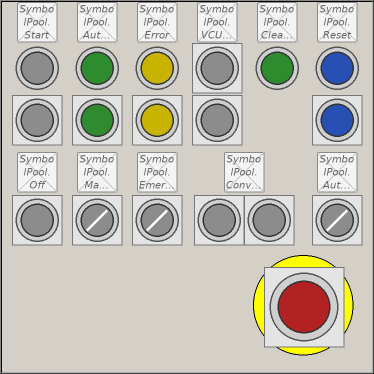
VISUALIZATION V_VC_AccessPanel  // 374x374
VAR_IN_OUT
	Signals : ST_VC_AccessPanel;
END_VAR
    Rectangle (0,0 374x374)
    Lamp1 (12,43 50x50), tooltip "Main contactor activeated", variable: Signals.outputs.LED_MainContactorActivated, style: Lamp-Lamp1-Gray
    PushSwitch (12,95 50x50), tooltip "Activate main contactor", variable: Signals.inputs.PB_ActivateMainContactor, behaviour: TAP, style: Switch-PushSwitch-Gray
    PushSwitch (72,95 50x50), tooltip "Auto on", variable: Signals.inputs.PB_AutoOn, behaviour: TAP, style: Switch-PushSwitch-Green
    Lamp1 (72,43 50x50), tooltip "Auto activated", variable: Signals.outputs.LED_AutoIsOn, style: Lamp-Lamp1-Green
    Lamp1 (132,43 50x50), tooltip "Error", variable: Signals.outputs.LED_Error, style: Lamp-Lamp1-Yellow
    PushSwitch (132,95 50x50), tooltip "Reset error", variable: Signals.inputs.PB_ErrorReset, behaviour: TAP, style: Switch-PushSwitch-Yellow
    RotarySwitch (72,195 50x50), tooltip "Man/Auto key switch", variable: Signals.inputs.SW_Auto, behaviour: TOGGLE, style: Switch-RotarySwitch-Gray
    PushSwitch (12,195 50x50), tooltip "Main contactor off", variable: Signals.inputs.PB_MainContactorOff, behaviour: TAP, style: Switch-PushSwitch-Gray
    Image (17,2 40x40), image: SymbolPool.Start
    Image (77,2 40x40), image: SymbolPool.AutoOn
    Image (137,2 40x40), image: SymbolPool.Error
    Image (17,152 40x40), image: SymbolPool.Off
    Image (77,152 40x40), image: SymbolPool.ManAuto
    Image (197,2 40x40), image: SymbolPool.VCUpDown
    PushSwitch (192,95 50x50), tooltip "VC Down", variable: Signals.inputs.PB_VcDown, behaviour: TAP, style: Switch-PushSwitch-Gray
    PushSwitch (192,43 50x50), tooltip "VC Up", variable: Signals.inputs.PB_VcUp, behaviour: TAP, style: Switch-PushSwitch-Gray
    Lamp1 (252,43 50x50), tooltip "Clear enterance", variable: Signals.outputs.LED_ClearEnterance, style: Lamp-Lamp1-Green
    Lamp1 (312,43 50x50), tooltip "Emergency stop", variable: Signals.outputs.LED_EmergencyStop, style: Lamp-Lamp1-Blue
    PushSwitch (312,95 50x50), tooltip "Reset emergency stop", variable: Signals.inputs.PB_EmergencyStopReset, behaviour: TAP, style: Switch-PushSwitch-Blue
    Image (257,2 40x40), image: SymbolPool.ClearToEnter
    Image (317,2 40x40), image: SymbolPool.Reset
    Image (224,152 40x40), image: SymbolPool.Conv_L_R
    PushSwitch (244,195 50x50), tooltip "VC Conveyor Right", variable: Signals.inputs.PB_VcConvRight, behaviour: TAP, style: Switch-PushSwitch-Gray
    PushSwitch (194,195 50x50), tooltip "VC Conveyor Left", variable: Signals.inputs.PB_VcConvLeft, behaviour: TAP, style: Switch-PushSwitch-Gray
    Image (317,152 40x40), image: SymbolPool.AutoMan
    RotarySwitch (312,195 50x50), tooltip "Auto/Entry request key switch", variable: Signals.inputs.SW_EntryRequest, behaviour: TOGGLE, style: Switch-RotarySwitch-Gray
    RotarySwitch (132,195 50x50), tooltip "Emergency drive key switch", variable: Signals.inputs.SW_EmergencyDrive, behaviour: TOGGLE, style: Switch-RotarySwitch-Gray
    Image (137,152 40x40), image: SymbolPool.EmergencyDrive
    Ellipse (253,255 100x100)
    PushSwitch (264,267 80x80), variable: Signals.inputs.PB_EmergencyStop, behaviour: TOGGLE, style: Switch-PushSwitch-Red
END_VISUALIZATION

(* stored: Version 1.1.0.1, ProductVersion 3.1.4024.9
   Visu V_VC_AccessPanel: Id {a7f34521-76ca-47b3-a23b-83fb7bd1f6cf} *)
